TYPE TcaStorageRef :
STRUCT
	Sensor AT%I* : BOOL;	
END_STRUCT
END_TYPE

(* stored: Version 1.1.0.1
   DUT TcaStorageRef: Id {1d2176cf-f7b9-498f-9094-be18690c5a22} *)
